TYPE ST_PodTelemetry :
    STRUCT
        // Mirrors the Rust struct in crates/protocol/src/lib.rs.
        // Wire layout: counter first (4 bytes LE), then timestamp (8 bytes LE).
        // Total payload size: 12 bytes.
        counter         : UDINT;    // u32, little-endian
        timestamp_us    : ULINT;    // u64, microseconds since some epoch
    END_STRUCT
END_TYPE

(* stored: Version 1.1.0.1
   DUT ST_PodTelemetry: Id {af5e9203-9ea2-4930-bb2a-ec026e9a0ede} *)
